FUNCTION FC_GetUsDateString : T_SHORT_STR;		// Returns the US date string, especially usefull for naming log files

FC_GetUsDateString := IING.usDateString;

END_FUNCTION

(* stored: Version 1.1.0.1, ProductVersion 3.1.4026.18
   POU FC_GetUsDateString: Id {ee2d7c63-2d2d-4b7d-b38f-a7b29f9738f3}, SpecialFunc None *)
